// LS Electric XG5000 project: fda
// PLC LSPLC
// module base 0 slot 0: 입출력 모듈:XBC-DR32H (DC 24V 입력, 릴레이 출력 32점)
// module base 0 slot 1: 위치결정 모듈:XBF-PD02A (위치결정 펄스(LD)출력형, 2축)
// module base 0 slot 2: 출력 모듈:XBE-TN/TP16A (트랜지스터 출력, 16점 (싱크출력/소스출력))

PROGRAM NewProgram (task: 스캔 프로그램)

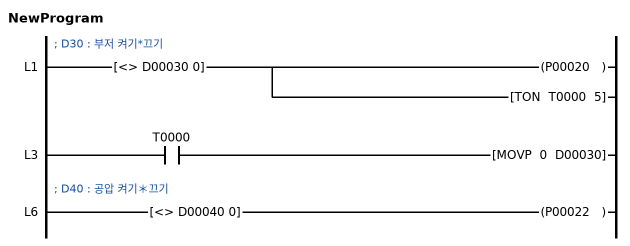
// D30 : 부저 켜기*끄기
; L1
LOAD<>    D00030 0
OUT       P00020
TON       T0000 5
; L3
LOAD      T0000
MOVP      0 D00030
// D40 : 공압 켜기＊끄기
; L6
LOAD<>    D00040 0
OUT       P00022